// Mitsubishi GX Works2 project: 機電整合丙級第二題-ST   PLC: FX3U/FX3UC

// task Task_01 (event TRUE, interval 0, priority 31): POU_01

PROGRAM POU_01
VAR
  wProgramStep : INT;
  tmT122 : TIME;
  tdT122 : TON;
  tmT22 : TIME;
  tdT22 : TON;
  tmT33 : TIME;
  tdT33 : TON;
  tmT23 : TIME;
  tdT23 : TON;
  tmT10 : TIME;
  tdT10 : TON;
  bM21 : BOOL;
  bM33 : BOOL;
  bM122 : BOOL;
  bM17 : BOOL;
  test : TIMER_100_FB_M;
END_VAR
(* 機電整合丙級術科第二題
   Author: Steven Luo
   Date: 2018/09/26
*)

IF M8002 OR NOT X17 THEN
	wProgramStep := 0;
	ZRST(TRUE, Y0, Y17);
	bM17 := FALSE;
	bM21 := FALSE;
	bM33 := FALSE;
	bM122 := FALSE;
END_IF;

IF NOT X17 THEN (* 按下急停 *)
	bM17 := TRUE;
END_IF;

IF X17 AND bM17 THEN (* 放開急停，等待復歸 *)
	wProgramStep := 122;
END_IF;

IF M8002 THEN
	wProgramStep := 21;
END_IF;

IF bM122 THEN
	IF M8013 THEN
		SET(TRUE, Y16); (* 黃燈閃爍 *)
	ELSE
		RST(TRUE, Y16);
	END_IF;
	tdT122(IN := TRUE, PT := T#3s); (* 計時三秒 *)
ELSE
	RST(TRUE, Y16);
END_IF;

IF (bM21 AND NOT bM33) OR (bM33 AND NOT M8013) THEN
	RST(TRUE, Y17); (*運轉中，綠燈滅、紅燈亮 *)
	SET(TRUE, Y15);
ELSE
	RST(TRUE, Y15); (* 待機，紅燈滅、綠燈亮 *)
	IF NOT bM17 AND NOT bM122 AND NOT M8013 THEN
		SET(TRUE, Y17);
	END_IF;
END_IF;

CASE wProgramStep OF
	21:
		IF X1 AND X3 AND X4 AND NOT X5 THEN
			IF X6 OR X7 THEN
				SET(TRUE, Y17); (* 待機，綠燈亮 *)
				bM122 := FALSE;
				bM21 := FALSE;
			END_IF;
		END_IF;
		IF X13 AND X17 AND X10 AND X16 THEN
			tdT122(IN := FALSE); (* tdT122的reset放在223似乎有問題，所以移到這裡 *)
			bM21 := TRUE; (* 工作模式、有料、按下啟動鈕 *)
			wProgramStep := 22;
		END_IF;
	22:
		tdT22(IN := X10, PT := T#3s); (* 計時三秒 *)
		IF tdT22.Q THEN
			IF X14 THEN (* 指定功能 *)
				wProgramStep := 33;
			ELSE (* 單一循環 *)
				IF X12 THEN
					bM33 := FALSE; (* 紅色料 *)
				ELSE
					bM33 := TRUE; (* 黑色料 *)
				END_IF;
				IF X11 THEN (* 開口朝上 *)
					wProgramStep := 26;
				ELSE (* 開口朝下 *)
					wProgramStep := 23;
				END_IF;
			END_IF;
			tdT22(IN := FALSE);
		END_IF;
	23:
		SET(TRUE, Y3); (* 夾爪夾料 *)
		tdT23(IN := TRUE, PT := T#1000ms); (* 計時一秒 *)
		IF tdT23.Q THEN
			SET(TRUE, Y0); (* 垂直剛上升 *)
			IF X0 THEN (* 垂直剛到達上端點 *)
				RST(TRUE, Y0);
				IF X6 THEN (* 迴轉馬達正轉端點 *)
					wProgramStep := 25;
				ELSIF X7 THEN (* 迴轉馬達反轉端點 *)
					wProgramStep := 35;
				END_IF;
			END_IF;
			tdT23(IN := FALSE);
		END_IF;
	25:
		SET(TRUE, Y7); (*迴轉馬達反轉 *)
		IF X7 THEN (* 迴轉馬達反轉端點 *)
			RST(TRUE, Y7);
			wProgramStep := 26;
		END_IF;
	26:
		SET(TRUE, Y1); (* 垂直剛下降 *)
		IF X1 THEN (* 垂直剛到達下端點 *)
			RST(TRUE, Y1);
			RST(TRUE, Y3);
			SET(TRUE, Y4); (* 夾爪放鬆 *)
			IF X4 THEN
				RST(TRUE, Y4);
				SET(TRUE, Y2); (* 迴轉缸至進料端 *)
				SET(X2, Y5); (* 吸盤吸 *)
			END_IF;
		END_IF;
		IF X5 THEN (* 真空壓力開關開 *)
			RST(TRUE, Y2); (* 迴轉缸至出料端 *)
			wProgramStep := 210;
		END_IF;
	33:
		bM33 := TRUE; (* 指定功能 *)
		SET(TRUE, Y3); (* 夾爪夾料 *)
		tdT33(IN := TRUE, PT := T#1000ms); (* 計時一秒 *)
		IF tdT33.Q THEN
			SET(TRUE, Y0); (* 垂直缸上升 *)
		END_IF;
		IF X0 THEN (* 垂直剛到達上端點 *)
			RST(TRUE, Y0);
			IF X6 THEN (* 迴轉馬達正轉端點 *)
				wProgramStep := 55;
			ELSIF X7 THEN (* 迴轉馬達反轉端點 *)
				wProgramStep := 56;
			END_IF;
			tdT33(IN := FALSE);
		END_IF;
	35:
		SET(TRUE, Y6); (* 迴轉馬達正轉 *)
		IF X6 THEN (* 迴轉馬達正轉端點 *)
			RST(TRUE, Y6);
			wProgramStep := 26;
		END_IF;
	55:
		SET(TRUE, Y7); (*迴轉馬達反轉 *)
		IF X7 THEN (* 迴轉馬達反轉端點 *)
			RST(TRUE, Y7);
			IF bM122 THEN
				wProgramStep := 125;
			ELSE
				wProgramStep := 66;
			END_IF;
		END_IF;
	56:
		SET(TRUE, Y6);; (* 迴轉馬達正轉 *)
		IF X6 THEN (* 迴轉馬達正轉端點 *)
			RST(TRUE, Y6);
			IF bM122 THEN
				wProgramStep := 125;
			ELSE
				wProgramStep := 66;
			END_IF;
		END_IF;
	66:
		SET(TRUE, Y1); (* 垂直剛下降 *)
		IF X1 THEN (* 垂直剛到達下端點 *)
			RST(TRUE, Y1);
			RST(TRUE, Y3);
			SET(TRUE, Y4); (* 夾爪放鬆 *)
			IF X4 THEN
				RST(TRUE, Y4);
				bM33 := FALSE;
				wProgramStep := 21;
			END_IF;
		END_IF;
	122:
		IF NOT X13 AND X16 THEN (* 復歸模式、按下復歸開關 *)
			bM122 := TRUE;
			bM17 := FALSE;
			IF NOT X4 THEN (*夾爪關 *)
				wProgramStep := 123;
			ELSE (*夾爪開 *)
				wProgramStep := 223;
			END_IF;
		END_IF;
	123:
		SET(TRUE, Y0); (* 垂直缸上升 *)
		IF X0 THEN (* 垂直剛到達上端點 *)
			RST(TRUE, Y0);
			IF X6 THEN (* 迴轉馬達正轉端點 *)
				wProgramStep := 55;
			ELSIF X7 THEN (* 迴轉馬達反轉端點 *)
				wProgramStep := 56;
			END_IF;
		END_IF;
	125:
		SET(TRUE, Y1); (* 垂直剛下降 *)
		IF X1 THEN (* 垂直剛到達下端點 *)
			RST(TRUE, Y1);
			SET(TRUE, Y4); (* 夾爪放鬆 *)
		END_IF;
		IF X4 AND tdT122.Q THEN
			RST(TRUE, Y4);
			wProgramStep := 21;
			tdT122(IN := FALSE);
			tdT22(IN := FALSE);
			tdT23(IN := FALSE);
			tdT33(IN := FALSE);
		END_IF;
	210:
		IF X3 THEN (* 迴轉缸至出料端 *)
			RST(TRUE, Y5);
			SET(TRUE, Y10); (* 真空吸盤放 *)
			IF NOT X5 THEN (* 真空壓力開關關 *)
				RST(TRUE, Y10);
				wProgramStep := 212;
			END_IF;
		END_IF;
	212:
		bM33 := FALSE;
		IF X15 THEN (* 連續循環 *)
			IF X10 THEN (* 有料 *)
				wProgramStep := 22;
			ELSE (* 無料 *)
				tdT10(IN := TRUE, PT := T#10s); (*計時十秒 *)
			END_IF;
			IF tdT10.Q THEN
				wProgramStep := 21; (* 十秒後回到待機狀態 *)
				tdT10(IN := FALSE);
			END_IF;
		ELSE
			wProgramStep := 21;
		END_IF;
	223:
		IF X3 THEN (* 迴轉缸至出料端 *)
			IF X5 THEN
				SET(TRUE, Y10); (* 真空吸盤放 *)
				IF NOT X5 THEN
					RST(TRUE, Y10);
				END_IF;
			END_IF;
			IF tdT122.Q THEN
				wProgramStep := 21;
(*				tdT122(IN := FALSE);*)
			END_IF;
		END_IF;
	ELSE
	;
END_CASE;
END_PROGRAM
